FUNCTION_BLOCK DIO_TRIGGERED_IN_8CH (* Service Interface Function Block Type *)
  (* Standard: 61499-2 *)
  (* Version 0.0, 16/09/2021, josef, nxtControl GmBH, template *)
  PACKAGE Flexbridge.Iceblock;
  (* Compiler Cpp nxtControl builtin 1.0 *)
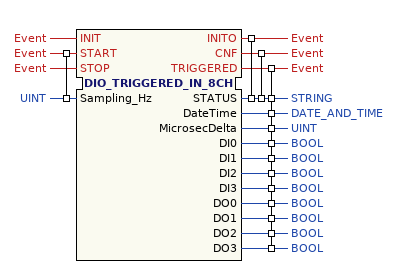
  EVENT_INPUT
    INIT; (* Service Initialization *)
    START WITH Sampling_Hz;
    STOP;
  END_EVENT
  EVENT_OUTPUT
    INITO WITH STATUS; (* Initialization Confirm *)
    CNF WITH STATUS;
    TRIGGERED WITH STATUS, DateTime, MicrosecDelta, DI0, DI1, DI2, DI3, DO0, DO1, DO2, DO3;
  END_EVENT
  VAR_INPUT
    Sampling_Hz : UINT := 1;
  END_VAR
  VAR_OUTPUT
    STATUS : STRING; (* Service Status *)
    DateTime : DATE_AND_TIME;
    MicrosecDelta : UINT;
    DI0 : BOOL;
    DI1 : BOOL;
    DI2 : BOOL;
    DI3 : BOOL;
    DO0 : BOOL;
    DO1 : BOOL;
    DO2 : BOOL;
    DO3 : BOOL;
  END_VAR
  SERVICE DIO_TRIGGERED_IN_4CH/RESOURCE
    SEQUENCE normal_establishment
      DIO_TRIGGERED_IN_4CH.INIT+(PARAMS) -> RESOURCE.initialize(PARAMS) -> DIO_TRIGGERED_IN_4CH.INITO+();
    END_SEQUENCE
    SEQUENCE unsuccessful_establishment
      DIO_TRIGGERED_IN_4CH.INIT+(PARAMS) -> RESOURCE.initialize(PARAMS) -> DIO_TRIGGERED_IN_4CH.INITO-(STATUS);
    END_SEQUENCE
    SEQUENCE request_confirm
      DIO_TRIGGERED_IN_4CH.REQ+(SD) -> RESOURCE.request(SD) -> DIO_TRIGGERED_IN_4CH.CNF+(RD);
    END_SEQUENCE
    SEQUENCE request_inhibited
      DIO_TRIGGERED_IN_4CH.REQ-(SD) -> DIO_TRIGGERED_IN_4CH.CNF-(STATUS);
    END_SEQUENCE
    SEQUENCE request_error
      DIO_TRIGGERED_IN_4CH.REQ+(SD) -> RESOURCE.request(SD) -> DIO_TRIGGERED_IN_4CH.CNF-(STATUS);
    END_SEQUENCE
    SEQUENCE indication_response
      RESOURCE.indicate(RD) -> DIO_TRIGGERED_IN_4CH.IND+(RD);
      DIO_TRIGGERED_IN_4CH.RSP(QI,SD) -> RESOURCE.response(QI,SD);
    END_SEQUENCE
    SEQUENCE indication_inhibited
      RESOURCE.indicate(RD,QI=FALSE) -> RESOURCE.inhibited();
    END_SEQUENCE
    SEQUENCE error_indication
      RESOURCE.error(STATUS) -> DIO_TRIGGERED_IN_4CH.IND-(STATUS);
    END_SEQUENCE
    SEQUENCE application_initiated_termination
      DIO_TRIGGERED_IN_4CH.INIT-() -> RESOURCE.terminate() -> DIO_TRIGGERED_IN_4CH.INITO-(STATUS);
    END_SEQUENCE
    SEQUENCE resource_initiated_termination
      -> DIO_TRIGGERED_IN_4CH.INITO-(STATUS);
    END_SEQUENCE
  END_SERVICE
END_FUNCTION_BLOCK
